    def rq_get_linear_axis_pos():
        axis_position = node_rpc_server.linearaxisgetactualposition()
        textmsg("Linear axis actual position : ", axis_position)
        return axis_position
    end
    global servojId = 2
  rq_collision_detection_stop()
  # end: URCap Installation Node
  global Waypoint_1_p=p[-.630407124235, -.296528896423, .136221788588, -1.229898520893, -1.220237997586, 1.196581871558]
  global Waypoint_1_q=[0.3692786395549774, -0.48095889509234624, 1.5607193152057093, 1.2628416258045654, -1.8477709929095667, -0.2628729979144495]
  global Waypoint_15_p=p[-.361117650575, -.287403925296, .558950815511, 1.229848458813, -1.214260238333, -1.194290411881]
  global Waypoint_15_q=[0.5462231636047363, -1.299070582990982, 1.9646461645709437, 1.6651934820362548, -1.9007957617389124, -0.3136795202838343]
  global Waypoint_16_p=p[-.635651184181, -.285475736443, .163792338200, -1.226772045383, -1.230615482384, 1.215161969706]
  global Waypoint_16_q=[0.33720043301582336, -0.5425684016994019, 1.5998790899859827, 1.293642206782959, -1.8175771872149866, -0.22054559389223272]
  global Waypoint_18_p=p[-.590750873318, -.139462379422, .307521318077, -1.226623837333, -1.230682192904, 1.215210985314]
  global Waypoint_18_q=[0.017998505383729935, -0.983365074997284, 2.003566090260641, 1.3587981897541503, -1.5887616316424769, 0.0046208566054701805]
  global Waypoint_19_p=p[-.489991526188, -.113644627590, .259460393076, 1.201174517973, 2.902848019224, .000152145723]
  global Waypoint_19_q=[-0.1367095152484339, -1.5985428295531214, 2.013503376637594, 3.7498223024555664, -0.966959301625387, -0.7424333731280726]
  global Waypoint_20_p=p[-.612491367170, -.235853461879, .172873629899, -.140583563832, 3.133080579292, -.008359806023]
  global Waypoint_20_q=[0.06762700862884163, -1.1663139852772701, 1.5767416058064176, 4.3262812889695015, -0.7725755715536655, -1.5973673863789557]
  global Waypoint_17_p=p[-.615869094666, .017644113422, .165499884759, -.140452718959, 3.133036764696, -.008284212182]
  global Waypoint_17_q=[-0.3403123060809534, -1.2111049455455323, 1.5604561010943812, 4.76623152473525, -0.8623440901385706, -2.1475346724139612]
  def calculate_point_to_move_towards(feature, direction, position_distance):
    local posDir=[direction[0], direction[1], direction[2]]
    if (norm(posDir) < 1e-6):
      return get_target_waypoint()
    end
    local direction_vector_normalized=normalize(posDir)
    local displacement_pose=p[direction_vector_normalized[0] * position_distance,direction_vector_normalized[1] * position_distance,direction_vector_normalized[2] * position_distance,0,0,0]
    local wanted_displacement_in_base_frame=pose_sub(pose_trans(feature, displacement_pose), feature)
    return pose_add(get_target_waypoint(), wanted_displacement_in_base_frame)
  end
  global Waypoint_31_p=p[-.620705477863, -.281438793834, .421856325693, .442241084011, -1.957788574586, 1.869446182328]
  global Waypoint_31_q=[-0.12204867998232061, -1.0642738503268738, 1.6338570753680628, 3.5765363413044433, 0.7937431335449219, -1.4932802359210413]
  global Waypoint_26_p=p[-.617598261035, -.285662220360, .447887815636, .257865385762, -2.080912438304, 2.083743282101]
  global Waypoint_26_q=[-0.11151010194887334, -1.1329282981208344, 1.640463654194967, 3.861135168666504, 0.8244242668151855, -1.443099323903219]
  global Waypoint_27_p=p[-.615450775964, -.280884121138, .196979310137, .186167416068, 2.228337584014, -2.171969679542]
  global Waypoint_27_q=[-0.1276615780040693, -0.8622460424642133, 1.8860316040763472, 3.7341520268710178, 0.7572025320077823, -1.4955693866647657]
  global Waypoint_30_p=p[-.495207212260, .028978859858, .374875227740, -1.178012939947, -1.429291973212, -1.137856928903]
  global Waypoint_30_q=[0.11711236089468002, -1.3994892698577424, 1.594299618397848, 0.04228417455639644, 2.3511312007904053, 1.775545358657837]
  global Waypoint_28_p=p[-.619839383396, .056782252985, .465016731825, -1.038625099662, -1.449976544355, -1.422633023255]
  global Waypoint_28_q=[0.05380272992719082, -1.049030689942267, 0.9311039597756929, 0.4607086029667755, 2.3871604587925592, 1.6100670367673615]
  global Waypoint_29_p=p[-.612286560883, .054274106350, .219229730051, -1.559816907949, -.273312861706, -.250072536663]
  global Waypoint_29_q=[0.054913531722276865, -0.9118303640193561, 1.8039951750427967, -2.1737980972152133, 2.382701554301983, 1.5099209384548118]
  global Waypoint_32_p=p[-.579373695775, -.099247829592, .329850635698, -1.080350767069, -1.256308939183, .949442715947]
  global Waypoint_32_q=[-0.0684283415423792, -1.6360942325987757, 2.298481289540426, -1.426223100428917, 1.424859881401062, 2.9433958530426025]
  global Waypoint_14_p=p[-.614394729902, -.211304335396, .158056240121, .891947218350, -1.398909790489, .897150739920]
  global Waypoint_14_q=[0.06688901782035828, -1.2062542003444214, 2.0273497740374964, -0.8648550671390076, 1.2756636142730713, -1.4902976194964808]
  global Waypoint_7_p=p[-.620397442971, -.213913387421, .513045981562, .892039726095, -1.398788049866, .897149319987]
  global Waypoint_7_q=[0.07276958227157593, -1.4890245211175461, 1.3829248587237757, 0.06161419927563472, 1.2746750116348267, -1.4881308714496058]
  global Waypoint_8_p=p[-.623058142139, -.006084652142, .504453333345, -1.537936671521, .945649868765, 1.518782592931]
  global Waypoint_8_q=[-0.19953567186464483, -1.5323755119792004, 1.506406609212057, 0.09952227651562495, 1.710647463798523, 1.639211893081665]
  global Waypoint_9_p=p[-.617185750904, -.003635744661, .159537482557, -1.537967820599, .945518640189, 1.518830856235]
  global Waypoint_9_q=[-0.2093423048602503, -1.1935233038714905, 2.0858619848834437, -0.8191923064044495, 1.7075483798980713, 1.6363801956176758]
  global Waypoint_11_p=p[-.622642705290, .073148999400, .262251367419, 2.006728907347, -1.984988481834, -.422320036043]
  global Waypoint_11_q=[-0.4727992403938508, -1.1931046923095465, 2.20874207186656, 2.5557256410267852, -1.073340525120777, -0.12859028859736554]
  global Waypoint_13_p=p[-.619354417627, -.281828120597, .259920784695, 2.006644977079, -1.985054067831, -.422363830708]
  global Waypoint_13_q=[0.34064259421721754, -1.0461214725192036, 1.9566921865069062, 2.624216301931531, -1.8247852350844171, 6.475282443617515]
  global Waypoint_10_p=p[-.530531214308, -.291051767939, .144441273867, -2.230084186391, -.010541297178, 2.193479360406]
  global Waypoint_10_q=[-0.013276402150289357, -1.1500203174403687, 2.071028534566061, -0.8113540571979065, 0.7900835871696472, 1.5619460344314575]
  global Waypoint_12_p=p[-.538683230436, -.290103741120, .513861909890, -2.230228499578, -.010549727182, 2.193403454803]
  global Waypoint_12_q=[-0.014661137257711232, -1.5093185876360913, 1.4554780165301722, 0.1618388134190063, 0.7814483642578125, 1.5644021034240723]
  global Waypoint_21_p=p[-.538097215403, -.306156956945, .483390788397, 1.229893655187, -1.218513911680, -1.215360660983]
  global Waypoint_21_q=[0.3963368409401085, -1.3775476134256621, 1.8729893210491355, -1.2799846272166313, 1.7980125332058048, 2.916890895394065]
  global Waypoint_22_p=p[-.536010150874, .078845475801, .482449152758, 1.229938842496, -1.218372029627, -1.215426474968]
  global Waypoint_22_q=[-0.5032866636859339, -1.6272269688048304, 2.161717716847555, -1.3892281365445633, 1.1609302759170532, 3.565915822982788]
  global Waypoint_23_p=p[-.536856714168, .057735272175, .516337801355, .007484190804, -1.587582998653, -.015116946919]
  global Waypoint_23_q=[-0.06483646191397252, -1.5618650824148386, 1.4615836328585363, 0.02914312769531069, 2.287159484941591, 4.71271091019117]
  global Waypoint_24_p=p[-.528032248544, .056709628722, .114658997919, .007476027220, -1.587403647508, -.015130351722]
  global Waypoint_24_q=[-0.06486922899355108, -1.1597505372813721, 2.1470850149737757, -1.0617385071567078, 2.2945711612701416, 4.708008766174316]
  global Waypoint_38_p=p[-.528301525964, .092928967835, .137544225611, 1.229518931609, -1.218164277810, -1.215725675197]
  global Waypoint_38_q=[-0.5465338865863245, -0.6870334309390564, 2.310338083897726, -2.490049978295797, 1.1306086778640747, 3.593946933746338]
  global Waypoint_25_p=p[-.530503307682, -.310799634742, .138539696150, 1.229529893186, -1.218212145518, -1.215748001331]
  global Waypoint_25_q=[0.4098140597343445, -0.6766109031489869, 2.0097950140582483, -2.1218296490111292, 1.8071534633636475, 2.900541067123413]
  global Waypoint_2_p=p[-.645397834819, -.296455318143, .135893598346, -1.229860133264, -1.220302156683, 1.196482482900]
  global Waypoint_2_q=[0.3583512306213379, -0.46596868455920415, 1.5182254950152796, 1.2925869661518554, -1.840168301259176, -0.25457460085024053]
  global Waypoint_3_p=p[-.653334935266, -.295509469566, .495795086421, -1.229748130315, -1.220382999730, 1.196524228234]
  global Waypoint_3_q=[0.3499549627304077, -1.030382589702942, 1.4344146887408655, 1.9436744886585693, -1.8333328405963343, -0.2433412710772913]
  global Waypoint_4_p=p[-.651378944197, .064515214832, .494965709811, -1.229676952695, -1.220192791007, 1.196530019033]
  global Waypoint_4_q=[-0.45318347612489873, -1.2302940350821991, 1.7351792494403284, 1.8209370809742431, -1.2614148298846644, 0.326932430267334]
  global Waypoint_5_p=p[-.643443913507, .063548429699, .135045355381, -1.229578554448, -1.220152089579, 1.196541404830]
  global Waypoint_5_q=[-0.45803863206972295, -0.5575369161418458, 1.8256614843951624, 1.0582493978687744, -1.2579148451434534, 0.32477086782455444]
  global Waypoint_6_p=p[-.645385399314, -.296430462109, .135967790852, -1.229561513341, -1.220089907423, 1.196571909520]
  global Waypoint_6_q=[0.3582976460456848, -0.4660030168345948, 1.5182111899005335, 1.2923266130634765, -1.8399995009051722, -0.25468570390810186]
  def sandRebate():
    $ 28 "sandRebate" "noBreak"
    $ 29 "MoveJ"
    $ 30 "Waypoint_16" "breakAfter"
    set_tcp(p[0.00318,0.11464,0.09820000000000001,-0.7853981633974483,0.0,0.0])
    movej(get_inverse_kin(pose_trans(CubeFront, pose_trans(p[.284950469331, -.169394328728, .660456967030, -1.179381585855, -1.206573510034, -1.222034237987], Waypoint_16_p)), qnear=Waypoint_16_q), a=1.3962634015954636, v=1.0471975511965976)
    $ 31 "Waypoint_18" "breakAfter"
    set_tcp(p[0.00318,0.11464,0.09820000000000001,-0.7853981633974483,0.0,0.0])
    movej(get_inverse_kin(pose_trans(CubeFront, pose_trans(p[.284950469331, -.169394328728, .660456967030, -1.179381585855, -1.206573510034, -1.222034237987], Waypoint_18_p)), qnear=Waypoint_18_q), a=1.3962634015954636, v=1.0471975511965976)
    $ 32 "Waypoint_19" "breakAfter"
    set_tcp(p[0.00318,0.11464,0.09820000000000001,-0.7853981633974483,0.0,0.0])
    movej(get_inverse_kin(pose_trans(CubeFront, pose_trans(p[.284950469331, -.169394328728, .660456967030, -1.179381585855, -1.206573510034, -1.222034237987], Waypoint_19_p)), qnear=Waypoint_19_q), a=1.3962634015954636, v=1.0471975511965976)
    $ 33 "Waypoint_20" "breakAfter"
    set_tcp(p[0.00318,0.11464,0.09820000000000001,-0.7853981633974483,0.0,0.0])
    movej(get_inverse_kin(pose_trans(CubeFront, pose_trans(p[.284950469331, -.169394328728, .660456967030, -1.179381585855, -1.206573510034, -1.222034237987], Waypoint_20_p)), qnear=Waypoint_20_q), a=1.3962634015954636, v=1.0471975511965976)
    # begin: URCap Program Node
    #   Source: Robotiq_Copilot, 1.22.1.14215, Robotiq Inc.
    #   Type: Find Surface
    $ 34 "Find Surface"
    zero_ftsensor()
    sleep(0.1)
    surface_found = rq_linear_search_urcap("Z+", 10.000, 0.005000, 0.100000, 1)
    storevar.setvariablepose("rq_findSurface_48dfa941-1460-4d19-a00f-d8f437f52397_exitPosition", get_actual_tcp_pose())
    $ 35 "'Add Stop conditions from the Find Surface node'" "noBreak"
    # 'Add Stop conditions from the Find Surface node'
    # end: URCap Program Node
    # begin: URCap Program Node
    #   Source: Robotiq_Copilot, 1.22.1.14215, Robotiq Inc.
    #   Type: Finishing Tool Control
    $ 36 "Start tool"
    set_standard_digital_out(3, True)
    # end: URCap Program Node
    $ 37 "Force"
    sleep(0.02)
    zero_ftsensor()
    force_mode(tool_pose(), [0, 0, 1, 0, 0, 0], [0.0, 0.0, 1.0, 0.0, 0.0, 0.0], 2, [0.1, 0.1, 0.15, 0.3490658503988659, 0.3490658503988659, 0.3490658503988659])
    $ 38 "MoveL" "noBreak"
    $ 39 "Waypoint_17" "noBreak"
    set_tcp(p[0.00318,0.11464,0.09820000000000001,-0.7853981633974483,0.0,0.0])
    movel(pose_trans(CubeFront, pose_trans(p[.284950469331, -.169394328728, .660456967030, -1.179381585855, -1.206573510034, -1.222034237987], Waypoint_17_p)), a=1.2, v=0.06)
    # begin: URCap Program Node
    #   Source: Robotiq_Copilot, 1.22.1.14215, Robotiq Inc.
    #   Type: Finishing Tool Control
    $ 40 "Stop tool" "noBreak"
    set_standard_digital_out(3, False)
    # end: URCap Program Node
    end_force_mode()
    stopl(5.0)
    $ 41 "MoveL"
    $ 42 "Direction: Tool Z-"
    global move_thread_flag_42=0
    thread move_thread_42():
      enter_critical
      move_thread_flag_42 = 1
      local towardsPos=calculate_point_to_move_towards(get_forward_kin(), [0.0,0.0,-1.0], 0.1)
      movel(towardsPos, a=1.2, v=0.25)
      move_thread_flag_42 = 2
      exit_critical
    end
    move_thread_flag_42 = 0
    move_thread_han_42 = run move_thread_42()
    while (True):
      sleep(1.0E-10)
      if (move_thread_flag_42 > 1):
        join move_thread_han_42
        $ 43 "Until (distance)"
        break
      end
      sync()
    end
    $ 44 "Direction: CubeFront Z+"
    global move_thread_flag_44=0
    thread move_thread_44():
      enter_critical
      move_thread_flag_44 = 1
      local towardsPos=calculate_point_to_move_towards(p[-0.6555216255462147,-0.29387207677313937,0.132153542128245,1.1865363507504816,1.2077692688007782,1.2289777735514902], [0.0,0.0,1.0], 0.15)
      movel(towardsPos, a=1.2, v=0.25)
      move_thread_flag_44 = 2
      exit_critical
    end
    move_thread_flag_44 = 0
    move_thread_han_44 = run move_thread_44()
    while (True):
      sleep(1.0E-10)
      if (move_thread_flag_44 > 1):
        join move_thread_han_44
        $ 45 "Until (distance)"
        break
      end
      sync()
    end
    $ 46 "MoveJ"
    $ 47 "Waypoint_31" "breakAfter"
    set_tcp(p[0.00318,0.11464,0.09820000000000001,-0.7853981633974483,0.0,0.0])
    movej(get_inverse_kin(pose_trans(CubeFront, pose_trans(p[.284950469331, -.169394328728, .660456967030, -1.179381585855, -1.206573510034, -1.222034237987], Waypoint_31_p)), qnear=Waypoint_31_q), a=1.3962634015954636, v=1.0471975511965976)
    $ 48 "Waypoint_26" "breakAfter"
    set_tcp(p[0.00318,0.11464,0.09820000000000001,-0.7853981633974483,0.0,0.0])
    movej(get_inverse_kin(pose_trans(CubeFront, pose_trans(p[.300286591152, -.149331691834, .650647942655, -1.193662016482, -1.190171861546, -1.213677846742], Waypoint_26_p)), qnear=Waypoint_26_q), a=1.3962634015954636, v=1.0471975511965976)
    # begin: URCap Program Node
    #   Source: Robotiq_Copilot, 1.22.1.14215, Robotiq Inc.
    #   Type: Find Surface
    $ 49 "Find Surface"
    zero_ftsensor()
    sleep(0.1)
    surface_found = rq_linear_search_urcap("Z+", 10.000, 0.005000, 0.100000, 1)
    storevar.setvariablepose("rq_findSurface_3ee7133c-89f8-43b4-bdcd-a21fe419666d_exitPosition", get_actual_tcp_pose())
    $ 50 "'Add Stop conditions from the Find Surface node'" "noBreak"
    # 'Add Stop conditions from the Find Surface node'
    # end: URCap Program Node
    # begin: URCap Program Node
    #   Source: Robotiq_Copilot, 1.22.1.14215, Robotiq Inc.
    #   Type: Finishing Tool Control
    $ 51 "Start tool"
    set_standard_digital_out(3, True)
    # end: URCap Program Node
    $ 52 "Force"
    sleep(0.02)
    zero_ftsensor()
    force_mode(tool_pose(), [0, 0, 1, 0, 0, 0], [0.0, 0.0, 1.0, 0.0, 0.0, 0.0], 2, [0.1, 0.1, 0.15, 0.3490658503988659, 0.3490658503988659, 0.3490658503988659])
    $ 53 "MoveL" "noBreak"
    $ 54 "Waypoint_27" "noBreak"
    set_tcp(p[0.00318,0.11464,0.09820000000000001,-0.7853981633974483,0.0,0.0])
    movel(pose_trans(CubeFront, pose_trans(p[.284950469331, -.169394328728, .660456967030, -1.179381585855, -1.206573510034, -1.222034237987], Waypoint_27_p)), a=1.2, v=0.06)
    # begin: URCap Program Node
    #   Source: Robotiq_Copilot, 1.22.1.14215, Robotiq Inc.
    #   Type: Finishing Tool Control
    $ 55 "Stop tool" "noBreak"
    set_standard_digital_out(3, False)
    # end: URCap Program Node
    end_force_mode()
    stopl(5.0)
    $ 56 "MoveL"
    $ 57 "Direction: Tool Z-"
    global move_thread_flag_57=0
    thread move_thread_57():
      enter_critical
      move_thread_flag_57 = 1
      local towardsPos=calculate_point_to_move_towards(get_forward_kin(), [0.0,0.0,-1.0], 0.05)
      movel(towardsPos, a=1.2, v=0.25)
      move_thread_flag_57 = 2
      exit_critical
    end
    move_thread_flag_57 = 0
    move_thread_han_57 = run move_thread_57()
    while (True):
      sleep(1.0E-10)
      if (move_thread_flag_57 > 1):
        join move_thread_han_57
        $ 58 "Until (distance)"
        break
      end
      sync()
    end
    $ 59 "Direction: CubeFront Z+"
    global move_thread_flag_59=0
    thread move_thread_59():
      enter_critical
      move_thread_flag_59 = 1
      local towardsPos=calculate_point_to_move_towards(p[-0.6555216255462147,-0.29387207677313937,0.132153542128245,1.1865363507504816,1.2077692688007782,1.2289777735514902], [0.0,0.0,1.0], 0.15)
      movel(towardsPos, a=1.2, v=0.25)
      move_thread_flag_59 = 2
      exit_critical
    end
    move_thread_flag_59 = 0
    move_thread_han_59 = run move_thread_59()
    while (True):
      sleep(1.0E-10)
      if (move_thread_flag_59 > 1):
        join move_thread_han_59
        $ 60 "Until (distance)"
        break
      end
      sync()
    end
    $ 61 "MoveJ"
    $ 62 "Waypoint_30" "breakAfter"
    set_tcp(p[0.00318,0.11464,0.09820000000000001,-0.7853981633974483,0.0,0.0])
    movej(get_inverse_kin(pose_trans(CubeFront, pose_trans(p[.284950469331, -.169394328728, .660456967030, -1.179381585855, -1.206573510034, -1.222034237987], Waypoint_30_p)), qnear=Waypoint_30_q), a=1.3962634015954636, v=1.0471975511965976)
    $ 63 "Waypoint_28" "breakAfter"
    set_tcp(p[0.00318,0.11464,0.09820000000000001,-0.7853981633974483,0.0,0.0])
    movej(get_inverse_kin(pose_trans(CubeFront, pose_trans(p[.284950469331, -.169394328728, .660456967030, -1.179381585855, -1.206573510034, -1.222034237987], Waypoint_28_p)), qnear=Waypoint_28_q), a=1.3962634015954636, v=1.0471975511965976)
    # begin: URCap Program Node
    #   Source: Robotiq_Copilot, 1.22.1.14215, Robotiq Inc.
    #   Type: Find Surface
    $ 64 "Find Surface"
    zero_ftsensor()
    sleep(0.1)
    surface_found = rq_linear_search_urcap("Z+", 10.000, 0.005000, 0.100000, 1)
    storevar.setvariablepose("rq_findSurface_0f0dcade-d478-4fc4-9bf8-a680beb3084f_exitPosition", get_actual_tcp_pose())
    $ 65 "'Add Stop conditions from the Find Surface node'" "noBreak"
    # 'Add Stop conditions from the Find Surface node'
    # end: URCap Program Node
    # begin: URCap Program Node
    #   Source: Robotiq_Copilot, 1.22.1.14215, Robotiq Inc.
    #   Type: Finishing Tool Control
    $ 66 "Start tool"
    set_standard_digital_out(3, True)
    # end: URCap Program Node
    $ 67 "Force"
    sleep(0.02)
    zero_ftsensor()
    force_mode(tool_pose(), [0, 0, 1, 0, 0, 0], [0.0, 0.0, 1.0, 0.0, 0.0, 0.0], 2, [0.1, 0.1, 0.15, 0.3490658503988659, 0.3490658503988659, 0.3490658503988659])
    $ 68 "MoveL" "noBreak"
    $ 69 "Waypoint_29" "noBreak"
    set_tcp(p[0.00318,0.11464,0.09820000000000001,-0.7853981633974483,0.0,0.0])
    movel(pose_trans(CubeFront, pose_trans(p[.284950469331, -.169394328728, .660456967030, -1.179381585855, -1.206573510034, -1.222034237987], Waypoint_29_p)), a=1.2, v=0.1)
    # begin: URCap Program Node
    #   Source: Robotiq_Copilot, 1.22.1.14215, Robotiq Inc.
    #   Type: Finishing Tool Control
    $ 70 "Stop tool" "noBreak"
    set_standard_digital_out(3, False)
    # end: URCap Program Node
    end_force_mode()
    stopl(5.0)
    $ 71 "MoveL"
    $ 72 "Direction: Tool Z-"
    global move_thread_flag_72=0
    thread move_thread_72():
      enter_critical
      move_thread_flag_72 = 1
      local towardsPos=calculate_point_to_move_towards(get_forward_kin(), [0.0,0.0,-1.0], 0.05)
      movel(towardsPos, a=1.2, v=0.25)
      move_thread_flag_72 = 2
      exit_critical
    end
    move_thread_flag_72 = 0
    move_thread_han_72 = run move_thread_72()
    while (True):
      sleep(1.0E-10)
      if (move_thread_flag_72 > 1):
        join move_thread_han_72
        $ 73 "Until (distance)"
        break
      end
      sync()
    end
    $ 74 "Direction: CubeFront Z+"
    global move_thread_flag_74=0
    thread move_thread_74():
      enter_critical
      move_thread_flag_74 = 1
      local towardsPos=calculate_point_to_move_towards(p[-0.6555216255462147,-0.29387207677313937,0.132153542128245,1.1865363507504816,1.2077692688007782,1.2289777735514902], [0.0,0.0,1.0], 0.15)
      movel(towardsPos, a=1.2, v=0.25)
      move_thread_flag_74 = 2
      exit_critical
    end
    move_thread_flag_74 = 0
    move_thread_han_74 = run move_thread_74()
    while (True):
      sleep(1.0E-10)
      if (move_thread_flag_74 > 1):
        join move_thread_han_74
        $ 75 "Until (distance)"
        break
      end
      sync()
    end
    $ 76 "MoveJ"
    $ 77 "Waypoint_32" "breakAfter"
    movej(get_inverse_kin(Waypoint_32_p, qnear=Waypoint_32_q), a=1.3962634015954636, v=1.0471975511965976)
  end
  def sprayRebate():
    $ 78 "sprayRebate" "noBreak"
    $ 79 "SprayRebate"
    $ 80 "MoveJ"
    $ 81 "Waypoint_14" "breakAfter"
    set_tcp(p[0.020839023181949995,-0.027139950822234082,0.10599373590389219,0.12258870209179472,1.1769383890382668,2.869747076630172])
    movej(get_inverse_kin(pose_trans(CubeFront, pose_trans(p[-.131847055554, -.113512547397, -.795239519450, .020655115358, .013310638043, -3.069721334155], Waypoint_14_p)), qnear=Waypoint_14_q), a=1.3962634015954636, v=1.0471975511965976)
    $ 82 "Set SprayerOn=On"
    set_standard_digital_out(5, True)
    $ 83 "MoveL"
    $ 84 "Waypoint_7" "breakAfter"
    movel(pose_trans(CubeFront, pose_trans(p[-.131847055554, -.113512547397, -.795239519450, .020655115358, .013310638043, -3.069721334155], Waypoint_7_p)), a=1.2, v=0.1)
    $ 85 "Set SprayerOn=Off"
    set_standard_digital_out(5, False)
    $ 86 "Direction: CubeFront Z+"
    global move_thread_flag_86=0
    thread move_thread_86():
      enter_critical
      move_thread_flag_86 = 1
      local towardsPos=calculate_point_to_move_towards(p[-0.6555216255462147,-0.29387207677313937,0.132153542128245,1.1865363507504816,1.2077692688007782,1.2289777735514902], [0.0,0.0,1.0], 0.1)
      movel(towardsPos, a=1.2, v=0.2)
      move_thread_flag_86 = 2
      exit_critical
    end
    move_thread_flag_86 = 0
    move_thread_han_86 = run move_thread_86()
    while (True):
      sleep(1.0E-10)
      if (move_thread_flag_86 > 1):
        join move_thread_han_86
        $ 87 "Until (distance)"
        break
      end
      sync()
    end
    $ 88 "MoveJ"
    $ 89 "Waypoint_8" "breakAfter"
    set_tcp(p[0.020839023181949995,-0.027139950822234082,0.10599373590389219,0.12258870209179472,1.1769383890382668,2.869747076630172])
    movej(get_inverse_kin(pose_trans(CubeFront, pose_trans(p[-.131847055554, -.113512547397, -.795239519450, .020655115358, .013310638043, -3.069721334155], Waypoint_8_p)), qnear=Waypoint_8_q), a=1.3962634015954636, v=1.0471975511965976)
    $ 90 "Set SprayerOn=On"
    set_standard_digital_out(5, True)
    $ 91 "MoveL"
    $ 92 "Waypoint_9" "breakAfter"
    set_tcp(p[0.020839023181949995,-0.027139950822234082,0.10599373590389219,0.12258870209179472,1.1769383890382668,2.869747076630172])
    movel(pose_trans(CubeFront, pose_trans(p[-.131847055554, -.113512547397, -.795239519450, .020655115358, .013310638043, -3.069721334155], Waypoint_9_p)), a=1.2, v=0.1)
    $ 93 "Set SprayerOn=Off"
    set_standard_digital_out(5, False)
    $ 94 "Direction: CubeFront Z+"
    global move_thread_flag_94=0
    thread move_thread_94():
      enter_critical
      move_thread_flag_94 = 1
      local towardsPos=calculate_point_to_move_towards(p[-0.6555216255462147,-0.29387207677313937,0.132153542128245,1.1865363507504816,1.2077692688007782,1.2289777735514902], [0.0,0.0,1.0], 0.1)
      movel(towardsPos, a=1.2, v=0.2)
      move_thread_flag_94 = 2
      exit_critical
    end
    move_thread_flag_94 = 0
    move_thread_han_94 = run move_thread_94()
    while (True):
      sleep(1.0E-10)
      if (move_thread_flag_94 > 1):
        join move_thread_han_94
        $ 95 "Until (distance)"
        break
      end
      sync()
    end
    $ 96 "MoveJ"
    $ 97 "Waypoint_11" "breakAfter"
    set_tcp(p[0.020839023181949995,-0.027139950822234082,0.10599373590389219,0.12258870209179472,1.1769383890382668,2.869747076630172])
    movej(get_inverse_kin(pose_trans(CubeFront, pose_trans(p[-.131847055554, -.113512547397, -.795239519450, .020655115358, .013310638043, -3.069721334155], Waypoint_11_p)), qnear=Waypoint_11_q), a=1.3962634015954636, v=1.0471975511965976)
    $ 98 "Set SprayerOn=On"
    set_standard_digital_out(5, True)
    $ 99 "MoveL"
    $ 100 "Waypoint_13" "breakAfter"
    set_tcp(p[0.020839023181949995,-0.027139950822234082,0.10599373590389219,0.12258870209179472,1.1769383890382668,2.869747076630172])
    movel(pose_trans(CubeFront, pose_trans(p[-.131847055554, -.113512547397, -.795239519450, .020655115358, .013310638043, -3.069721334155], Waypoint_13_p)), a=1.2, v=0.1)
    $ 101 "Set SprayerOn=Off"
    set_standard_digital_out(5, False)
    $ 102 "Direction: CubeFront Z+"
    global move_thread_flag_102=0
    thread move_thread_102():
      enter_critical
      move_thread_flag_102 = 1
      local towardsPos=calculate_point_to_move_towards(p[-0.6555216255462147,-0.29387207677313937,0.132153542128245,1.1865363507504816,1.2077692688007782,1.2289777735514902], [0.0,0.0,1.0], 0.1)
      movel(towardsPos, a=1.2, v=0.2)
      move_thread_flag_102 = 2
      exit_critical
    end
    move_thread_flag_102 = 0
    move_thread_han_102 = run move_thread_102()
    while (True):
      sleep(1.0E-10)
      if (move_thread_flag_102 > 1):
        join move_thread_han_102
        $ 103 "Until (distance)"
        break
      end
      sync()
    end
  end
  def sprayFront():
    $ 104 "sprayFront" "noBreak"
    $ 105 "SprayFront"
    $ 106 "MoveJ"
    $ 107 "Waypoint_10" "breakAfter"
    set_tcp(p[0.020839023181949995,-0.027139950822234082,0.10599373590389219,0.12258870209179472,1.1769383890382668,2.869747076630172])
    movej(get_inverse_kin(pose_trans(CubeFront, pose_trans(p[-.131847055554, -.113512547397, -.795239519450, .020655115358, .013310638043, -3.069721334155], Waypoint_10_p)), qnear=Waypoint_10_q), a=1.3962634015954636, v=1.0471975511965976)
    $ 108 "Set SprayerOn=On"
    set_standard_digital_out(5, True)
    $ 109 "MoveL"
    $ 110 "Waypoint_12" "breakAfter"
    movel(pose_trans(CubeFront, pose_trans(p[-.131847055554, -.113512547397, -.795239519450, .020655115358, .013310638043, -3.069721334155], Waypoint_12_p)), a=1.2, v=0.1)
    $ 111 "Set SprayerOn=Off"
    set_standard_digital_out(5, False)
    $ 112 "Direction: Tool Z-"
    global move_thread_flag_112=0
    thread move_thread_112():
      enter_critical
      move_thread_flag_112 = 1
      local towardsPos=calculate_point_to_move_towards(get_forward_kin(), [0.0,0.0,-1.0], 0.1)
      movel(towardsPos, a=1.2, v=0.2)
      move_thread_flag_112 = 2
      exit_critical
    end
    move_thread_flag_112 = 0
    move_thread_han_112 = run move_thread_112()
    while (True):
      sleep(1.0E-10)
      if (move_thread_flag_112 > 1):
        join move_thread_han_112
        $ 113 "Until (distance)"
        break
      end
      sync()
    end
    $ 114 "MoveJ"
    $ 115 "Waypoint_21" "breakAfter"
    set_tcp(p[0.020839023181949995,-0.027139950822234082,0.10599373590389219,0.12258870209179472,1.1769383890382668,2.869747076630172])
    movej(get_inverse_kin(pose_trans(CubeFront, pose_trans(p[-.131847055554, -.113512547397, -.795239519450, .020655115358, .013310638043, -3.069721334155], Waypoint_21_p)), qnear=Waypoint_21_q), a=1.3962634015954636, v=1.0471975511965976)
    $ 116 "Set SprayerOn=On"
    set_standard_digital_out(5, True)
    $ 117 "MoveL"
    $ 118 "Waypoint_22" "breakAfter"
    set_tcp(p[0.020839023181949995,-0.027139950822234082,0.10599373590389219,0.12258870209179472,1.1769383890382668,2.869747076630172])
    movel(pose_trans(CubeFront, pose_trans(p[-.131847055554, -.113512547397, -.795239519450, .020655115358, .013310638043, -3.069721334155], Waypoint_22_p)), a=1.2, v=0.1)
    $ 119 "Set SprayerOn=Off"
    set_standard_digital_out(5, False)
    $ 120 "Direction: Tool Z-"
    global move_thread_flag_120=0
    thread move_thread_120():
      enter_critical
      move_thread_flag_120 = 1
      local towardsPos=calculate_point_to_move_towards(get_forward_kin(), [0.0,0.0,-1.0], 0.1)
      movel(towardsPos, a=1.2, v=0.2)
      move_thread_flag_120 = 2
      exit_critical
    end
    move_thread_flag_120 = 0
    move_thread_han_120 = run move_thread_120()
    while (True):
      sleep(1.0E-10)
      if (move_thread_flag_120 > 1):
        join move_thread_han_120
        $ 121 "Until (distance)"
        break
      end
      sync()
    end
    $ 122 "MoveJ"
    $ 123 "Waypoint_23" "breakAfter"
    set_tcp(p[0.020839023181949995,-0.027139950822234082,0.10599373590389219,0.12258870209179472,1.1769383890382668,2.869747076630172])
    movej(get_inverse_kin(pose_trans(CubeFront, pose_trans(p[-.131847055554, -.113512547397, -.795239519450, .020655115358, .013310638043, -3.069721334155], Waypoint_23_p)), qnear=Waypoint_23_q), a=1.3962634015954636, v=1.0471975511965976)
    $ 124 "Set SprayerOn=On"
    set_standard_digital_out(5, True)
    $ 125 "MoveL"
    $ 126 "Waypoint_24" "breakAfter"
    set_tcp(p[0.020839023181949995,-0.027139950822234082,0.10599373590389219,0.12258870209179472,1.1769383890382668,2.869747076630172])
    movel(pose_trans(CubeFront, pose_trans(p[-.131847055554, -.113512547397, -.795239519450, .020655115358, .013310638043, -3.069721334155], Waypoint_24_p)), a=1.2, v=0.1)
    $ 127 "Set SprayerOn=Off"
    set_standard_digital_out(5, False)
    $ 128 "Direction: Tool Z-"
    global move_thread_flag_128=0
    thread move_thread_128():
      enter_critical
      move_thread_flag_128 = 1
      local towardsPos=calculate_point_to_move_towards(get_forward_kin(), [0.0,0.0,-1.0], 0.1)
      movel(towardsPos, a=1.2, v=0.2)
      move_thread_flag_128 = 2
      exit_critical
    end
    move_thread_flag_128 = 0
    move_thread_han_128 = run move_thread_128()
    while (True):
      sleep(1.0E-10)
      if (move_thread_flag_128 > 1):
        join move_thread_han_128
        $ 129 "Until (distance)"
        break
      end
      sync()
    end
    $ 130 "MoveJ"
    $ 131 "Waypoint_38" "breakAfter"
    set_tcp(p[0.020839023181949995,-0.027139950822234082,0.10599373590389219,0.12258870209179472,1.1769383890382668,2.869747076630172])
    movej(get_inverse_kin(pose_trans(CubeFront, pose_trans(p[-.131847055554, -.113512547397, -.795239519450, .020655115358, .013310638043, -3.069721334155], Waypoint_38_p)), qnear=Waypoint_38_q), a=1.3962634015954636, v=1.0471975511965976)
    $ 132 "Set SprayerOn=On"
    set_standard_digital_out(5, True)
    $ 133 "MoveL"
    $ 134 "Waypoint_25" "breakAfter"
    set_tcp(p[0.020839023181949995,-0.027139950822234082,0.10599373590389219,0.12258870209179472,1.1769383890382668,2.869747076630172])
    movel(pose_trans(CubeFront, pose_trans(p[-.131847055554, -.113512547397, -.795239519450, .020655115358, .013310638043, -3.069721334155], Waypoint_25_p)), a=1.2, v=0.1)
    $ 135 "Set SprayerOn=Off"
    set_standard_digital_out(5, False)
    $ 136 "Direction: Tool Z-"
    global move_thread_flag_136=0
    thread move_thread_136():
      enter_critical
      move_thread_flag_136 = 1
      local towardsPos=calculate_point_to_move_towards(get_forward_kin(), [0.0,0.0,-1.0], 0.1)
      movel(towardsPos, a=1.2, v=0.2)
      move_thread_flag_136 = 2
      exit_critical
    end
    move_thread_flag_136 = 0
    move_thread_han_136 = run move_thread_136()
    while (True):
      sleep(1.0E-10)
      if (move_thread_flag_136 > 1):
        join move_thread_han_136
        $ 137 "Until (distance)"
        break
      end
      sync()
    end
  end
  def sandFront():
    $ 138 "sandFront" "noBreak"
    $ 139 "sandFront"
    $ 140 "Set"
    set_tcp(p[0.00318,0.11464,0.09820000000000001,-0.7853981633974483,0.0,0.0])
    $ 141 "MoveL"
    $ 142 "Waypoint_2" "breakAfter"
    set_tcp(p[0.00318,0.11464,0.09820000000000001,-0.7853981633974483,0.0,0.0])
    movel(pose_trans(CubeFront, pose_trans(p[-.131847055554, -.113512547397, -.795239519450, .020655115358, .013310638043, -3.069721334155], Waypoint_2_p)), a=1.2, v=0.25)
    # begin: URCap Program Node
    #   Source: Robotiq_Copilot, 1.22.1.14215, Robotiq Inc.
    #   Type: Zero FT Sensor
    $ 143 "Zero FT Sensor"

    rq_wait_ft_sensor_steady(2000)
    zero_ftsensor()
    sleep(0.1)
    # end: URCap Program Node
    $ 144 "Direction: Tool Z+"
    global move_thread_flag_144=0
    thread move_thread_144():
      enter_critical
      move_thread_flag_144 = 1
      local towardsPos=calculate_point_to_move_towards(get_forward_kin(), [0.0,0.0,1.0], 1000.0)
      movel(towardsPos, a=1.2, v=0.05)
      move_thread_flag_144 = 2
      exit_critical
    end
    move_thread_flag_144 = 0
    move_thread_han_144 = run move_thread_144()
    while (True):
      local targetTcpDirection=get_target_tcp_speed()
      local stepsToRetract=tool_contact(direction=targetTcpDirection)
      if (stepsToRetract > 0):
        kill move_thread_han_144
        stopl(3.0)
        $ 145 "Until (tool_contact_detection)"
        break
      end
      sync()
    end
    # begin: URCap Program Node
    #   Source: Robotiq_Copilot, 1.22.1.14215, Robotiq Inc.
    #   Type: Finishing Tool Control
    $ 146 "Start tool"
    set_standard_digital_out(3, True)
    # end: URCap Program Node
    $ 147 "Wait: 1.0"
    sleep(1.0)
    $ 148 "MoveL"
    # begin: URCap Program Node
    #   Source: Robotiq_Copilot, 1.22.1.14215, Robotiq Inc.
    #   Type: Zero FT Sensor
    $ 149 "Zero FT Sensor"

    zero_ftsensor()
    sleep(0.1)
    # end: URCap Program Node
    $ 150 "Force"
    sleep(0.02)
    zero_ftsensor()
    force_mode(tool_pose(), [0, 0, 1, 0, 0, 0], [0.0, 0.0, 1.0, 0.0, 0.0, 0.0], 2, [0.1, 0.1, 0.15, 0.3490658503988659, 0.3490658503988659, 0.3490658503988659])
    $ 151 "Waypoint_3" "noBreak"
    set_tcp(p[0.00318,0.11464,0.09820000000000001,-0.7853981633974483,0.0,0.0])
    movel(pose_trans(CubeFront, pose_trans(p[-.131847055554, -.113512547397, -.795239519450, .020655115358, .013310638043, -3.069721334155], Waypoint_3_p)), a=1.2, v=0.12)
    $ 152 "Waypoint_4" "noBreak"
    set_tcp(p[0.00318,0.11464,0.09820000000000001,-0.7853981633974483,0.0,0.0])
    movel(pose_trans(CubeFront, pose_trans(p[-.131847055554, -.113512547397, -.795239519450, .020655115358, .013310638043, -3.069721334155], Waypoint_4_p)), a=1.2, v=0.12)
    $ 153 "Waypoint_5" "noBreak"
    set_tcp(p[0.00318,0.11464,0.09820000000000001,-0.7853981633974483,0.0,0.0])
    movel(pose_trans(CubeFront, pose_trans(p[-.131847055554, -.113512547397, -.795239519450, .020655115358, .013310638043, -3.069721334155], Waypoint_5_p)), a=1.2, v=0.12)
    $ 154 "Waypoint_6" "noBreak"
    set_tcp(p[0.00318,0.11464,0.09820000000000001,-0.7853981633974483,0.0,0.0])
    movel(pose_trans(CubeFront, pose_trans(p[-.131847055554, -.113512547397, -.795239519450, .020655115358, .013310638043, -3.069721334155], Waypoint_6_p)), a=1.2, v=0.12)
    # begin: URCap Program Node
    #   Source: Robotiq_Copilot, 1.22.1.14215, Robotiq Inc.
    #   Type: Finishing Tool Control
    $ 155 "Stop tool" "noBreak"
    set_standard_digital_out(3, False)
    # end: URCap Program Node
    end_force_mode()
    stopl(5.0)
    $ 156 "Direction: Tool Z-"
    global move_thread_flag_156=0
    thread move_thread_156():
      enter_critical
      move_thread_flag_156 = 1
      local towardsPos=calculate_point_to_move_towards(get_forward_kin(), [0.0,0.0,-1.0], 0.025)
      movel(towardsPos, a=1.2, v=0.12)
      move_thread_flag_156 = 2
      exit_critical
    end
    move_thread_flag_156 = 0
    move_thread_han_156 = run move_thread_156()
    while (True):
      sleep(1.0E-10)
      if (move_thread_flag_156 > 1):
        join move_thread_han_156
        $ 157 "Until (distance)"
        break
      end
      sync()
    end
  end
  thread EventThread():
    while (True):
      if (get_standard_digital_in(2) ==   True  ):
        $ 14 "Set ClampOn=On"
        set_standard_digital_out(7, True)
        $ 15 "MoveJ"
        $ 16 "Waypoint_1" "breakAfter"
        set_tcp(p[0.00318,0.11464,0.09820000000000001,-0.7853981633974483,0.0,0.0])
        movej(get_inverse_kin(pose_trans(CubeFront, pose_trans(p[.300286591152, -.149331691834, .650647942655, -1.193662016482, -1.190171861546, -1.213677846742], Waypoint_1_p)), qnear=Waypoint_1_q), a=1.3962634015954636, v=1.0471975511965976)
        $ 17 "Call sandFront"
        sandFront()
        $ 18 "Call sandFront"
        sandFront()
        $ 21 "MoveJ"
        $ 22 "Waypoint_1" "breakAfter"
        set_tcp(p[0.00318,0.11464,0.09820000000000001,-0.7853981633974483,0.0,0.0])
        movej(get_inverse_kin(pose_trans(CubeFront, pose_trans(p[.300286591152, -.149331691834, .650647942655, -1.193662016482, -1.190171861546, -1.213677846742], Waypoint_1_p)), qnear=Waypoint_1_q), a=1.3962634015954636, v=1.0471975511965976)
        $ 23 "Call sprayFront"
        sprayFront()
        $ 24 "Call sprayRebate"
        sprayRebate()
        $ 25 "Set ClampOn=Off"
        set_standard_digital_out(7, False)
        $ 26 "MoveJ"
        $ 27 "Waypoint_15" "breakAfter"
        set_tcp(p[0.020839023181949995,-0.027139950822234082,0.10599373590389219,0.12258870209179472,1.1769383890382668,2.869747076630172])
        movej(get_inverse_kin(Waypoint_15_p, qnear=Waypoint_15_q), a=1.3962634015954636, v=1.0471975511965976)
      end
      sync()
    end
  end
  eventThread = run EventThread()
  while (True):
    $ 1 "Robot Program"
    $ 2 "Set PinsUp=On"
    set_standard_digital_out(6, True)
    $ 3 "Wait: 0.01"
    sleep(0.01)
  end
end
